TEXTLIST tlHPv3
  1 = 'M1- Inner - Outer Cap'
  2 = 'M2- Mug - Outer Cap'
  3 = 'M3- Mug - Bayonet'
  0 = 'HotPlate nest, station %s' | pl: 'Gniazdo HotPlate, stacja %s'
  10 = 'Initialization' | pl: 'Inicjalizacja'
  11 = 'Manual work' | pl: 'Praca ręczna'
  12 = 'Ready for new operation' | pl: 'Gotowy/a na nową operację'
  13 = 'Performing reference weld' | pl: 'Przeprowadzanie zgrzewu referencyjnego'
  14 = 'Measure Axis distance' | pl: 'Pomiar odległości napędów'
  15 = 'Measure Heated Plate Height' | pl: 'Pomiar wysokości płyty grzejnej'
  16 = 'Welding in progress' | pl: 'Trwa operacja zgrzewania'
  17 = 'ERROR ACTIVE' | pl: 'BŁĄD AKTYWNY'
  19 = 'Moving to safe state' | pl: 'Jazda do pozycji bezpiecznej'
  20 = 'Error, waiting for confirmation' | pl: 'Błąd, oczekiwanie na potwierdzenie'
  21 = 'Reset machine to base state' | pl: 'Reset maszyny do pozycji bazowej'
  22 = 'Moving to Pre-Base position' | pl: 'Jzda do pozycji pre-bazowej'
  23 = 'Adjustment start delay (for simultanously departure)' | pl: 'Opóźnienie startu dopasowania (jednoczesny odjazd)'
  24 = 'Adjustment in progress' | pl: 'Dopasowanie części'
  25 = 'Parts heatup' | pl: 'Nagrzewanie części'
  26 = 'Part heatedup - wait for departure permission' | pl: 'Część nagrzana- oczekiwanie na odjazd'
  27 = 'Departure from HeatedPlate' | pl: 'Odjazd od płyty grzejnej'
  28 = 'Wait for hide HeatedPlate' | pl: 'Oczekiwanie na schowanie płyty grzejnej'
  29 = 'Moving to connection point' | pl: 'Jazda do punktu łączenia'
  30 = 'Connecting in progress' | pl: 'Łączenie części'
  31 = 'Cooling down parts after connection' | pl: 'Studzenie części po zgrzewie'
  32 = 'New operation in progress' | pl: 'Trwa nowa operacja'
  33 = 'Part marking' | pl: 'Znakowanie części'
  34 = 'Return to base state' | pl: 'Powrót do stanu domyślnego'
  35 = 'Wait for insert calibration templates into clamps and close workcover' | pl: 'Oczekiwanie na montaż wzorców kalibracyjnych oraz zamknięcie osłony'
  36 = 'Time for remove calibration templates and save or not results' | pl: 'Usuwanie wzorców kalib. oraz zapis lub nie wyników pomiaru'
   = ''
END_TEXTLIST

(* stored: Version 1.1.0.1, ProductVersion 3.1.4024.12
   TextList tlHPv3: Id {45558fb8-7f1c-4fad-bdce-613b50ca059c} *)
